(* IEC 61131-3 sources: CodesysTest/export/SX_1195.dev/Plc Logic/Application/PRJ Specific/Motion/Motors/Oriental AZD/AZD-KR2D/FB_OrientalAZMotorTriggerPositionTest.pou, 3 files *)

(* ---- FB_OrientalAZMotorTriggerPositionTest.pou.st ---- *)
(*#-#-#-#-#-#-#-#-#-#---Declaration---#-#-#-#-#-#-#-#-#-#-#-#-#*)

FUNCTION_BLOCK FB_OrientalAZMotorTriggerPositionTest EXTENDS Axis_REF
VAR_INPUT
	// Set this flag if this motor is actually a group
	isGroup : BOOL;
	// Steps per inch of motion
	stepsPerInchSP : DINT := 3999;
	// At factory "zero" there can be an offset
	zeroOffset : REAL;
	// Jog motor forward command
	jogForwardCMD : BOOL;
	// Jog motor reverse command
	jogReverseCMD : BOOL;
	// Factory "zero" positon preset command
	positionPresetRequest : BOOL;
	// Free up motor command
	freeMotorRequest : BOOL;
	// Ref to Master Motor if group
	groupMotor0 : REFERENCE TO FB_OrientalAZMotorTriggerPositionTest;
	// Ref to Slave Motor if group
	groupMotor1 : REFERENCE TO FB_OrientalAZMotorTriggerPositionTest;
END_VAR
VAR_OUTPUT
	// Hex alarm code reported from AZ Drive
	alarmCode : DWORD;
	// Trigger direct data write through modbus
	triggerDDWriteNow : BOOL;
	// Trigger Remote I/O data write through modbus
	triggerRIOWriteNow : BOOL;
END_VAR
VAR
	directDataOp : sctOrientalDirectData;
	distanceFromDrive : uModbusDWORD;
	alarmCodeFromDrive : uModbusDWORD;
	ready : BOOL;
	alarmActive : BOOL;
	moving : BOOL;
	inPosition : BOOL;
	atTorqueLimit : BOOL;
	atPosition : BOOL;
	homeSwitchTrigger : BOOL;
	homeNow : BOOL;
	P_Preset : BOOL;
	start : BOOL;
	zHome : BOOL;
	stop : BOOL;
	freeMotor : BOOL;
	reset : BOOL;
	EL_Preset : BOOL;
	jogReverse : BOOL;
	jogForward : BOOL;
	packedRIO : uModbusDWORD;
	packedRIOLast : DWORD;
	delayTimer : Standard.TON := (PT := T#50MS);
	zHomeDelay : Standard.TON := (PT := T#250MS);
	presetDelay : Standard.TON := (PT := T#200MS);
	modbusWriteResponse : ARRAY[0..20] OF WORD;
	readAfterDDWrite : FB_ONS;
	readAfterRIOWrite : FB_ONS;
	triggerPositonPreset : FB_ONS;
	haltONS : FB_ONS;
	alarmActiveONS : FB_ONS;
	freeMotorRequestONS : FB_ONS;
	triggerRIOWrite : BOOL;
	resetRIOWrite : Standard.TON := (PT := T#50MS);
	disable : BOOL;
	enumAlarmCode : eOrientalAZDriveFaults;
	state : eOrientalAZDriveStates;
	nextState : eOrientalAZDriveStates;
	commErrorONS : FB_ONS;
	commErrorFaultONS : FB_ONS;
	commErrorCount : DINT;
	commErrorFaultSetting : DINT := 3;
	positionPresetONS : FB_ONS;
END_VAR
VAR_IN_OUT
	MBChannel : IoDrvModbus.ModbusSlaveComPort;
	modbusDataFromDrive : ARRAY[0..39] OF WORD;
	modbusDirectDataToDrive : ARRAY[0..16] OF WORD;
	modbusRIODataToDrive : ARRAY[0..1] OF WORD;
END_VAR(*#-#-#-#-#-#-#-#-#-#---Implementation---#-#-#-#-#-#-#-#-#-#-#-#-#*)

//	Function Block: FB_OrientalAZMotor()
//	Description: A PLCOpen Motion compliant library for a Oriental AZ Series drive/motor
//
//	Created by: Ben Hess
//	Created Date: Tuesday, June 2nd 2020

// Outputs for Motion Lib
operational := PowerOn;
EnableState := DriveEnable;

// Exit if drive isn't enabled.
IF NOT DriveEnable THEN
	Error := FALSE;
	RETURN;
END_IF

// Get raw drive position and alarm code
IF isGroup THEN
	IF __ISVALIDREF(groupMotor0) THEN
		actPos := groupMotor0.ActualPosition;
		enumAlarmCode := groupMotor0.enumAlarmCode;
	END_IF
ELSE
	distanceFromDrive.wWord[0] := modbusDataFromDrive[3];
	distanceFromDrive.wWord[1] := modbusDataFromDrive[2];
	actPos := (TO_REAL(distanceFromDrive.diDint) / TO_REAL(stepsPerInchSP)) + zeroOffset;
	alarmCodeFromDrive.wWord[0] := modbusDataFromDrive[7];
	alarmCodeFromDrive.wWord[1] := modbusDataFromDrive[6];
	enumAlarmCode := TO_INT(alarmCodeFromDrive.diDint);
END_IF
alarmCode := TO_DWORD(enumAlarmCode);

// Pack RIO to write to drive
packedRIO.dDword.0 := homeSwitchTrigger;
packedRIO.dDword.1 := homeNow;
packedRIO.dDword.2 := P_Preset;
packedRIO.dDword.3 := start;
packedRIO.dDword.4 := zHome;
packedRIO.dDword.5 := stop;
packedRIO.dDword.6 := freeMotor;
packedRIO.dDword.7 := reset;
packedRIO.dDword.12 := EL_Preset;
packedRIO.dDword.13 := jogReverse;
packedRIO.dDword.14 := jogForward;
modbusRIODataToDrive[0] := packedRIO.wWord[1];
modbusRIODataToDrive[1] := packedRIO.wWord[0];

// Setup delay timers
delayTimer(IN := state = eOrientalAZDriveStates.DelayAfterWrite);
zHomeDelay(IN := state = eOrientalAZDriveStates.Homing);
presetDelay(IN := state = eOrientalAZDriveStates.SettingPreset);
// Trigger an RIO write whenever it changes
IF packedRIO.dDword <> packedRIOLast AND NOT triggerRIOWriteNow THEN
	packedRIOLast := packedRIO.dDword;
	triggerRIOWriteNow := TRUE;
END_IF
resetRIOWrite(IN := triggerRIOWriteNow);
IF resetRIOWrite.Q THEN
	triggerRIOWriteNow := FALSE;
END_IF
positionPresetONS(CLK := positionPresetRequest);

// Only set comm error status after x modbus errors
commErrorONS(CLK := MBChannel.xError);
IF commErrorONS.OSR THEN
	commErrorCount := commErrorCount + 1;
END_IF
commErrorFaultONS(CLK := commErrorCount = commErrorFaultSetting);
IF NOT isGroup THEN
	IF commErrorFaultONS.OSR THEN
		state := eOrientalAZDriveStates.Faulting;
		CommStatus := FALSE;
	END_IF
END_IF

// Get drive data directly from modbus or from master axis
IF isGroup THEN
	IF __ISVALIDREF(groupMotor0) AND __ISVALIDREF(groupMotor1) THEN
		ready := groupMotor0.ready AND groupMotor1.ready;
		alarmActive := groupMotor0.alarmActive OR groupMotor1.alarmActive;
		moving := groupMotor0.moving AND groupMotor1.moving;
		inPosition := groupMotor0.inPosition AND groupMotor1.inPosition;
		atTorqueLimit := groupMotor0.atTorqueLimit OR groupMotor1.atTorqueLimit;
	END_IF
ELSE
	Ready := modbusDataFromDrive[5].5;
	AlarmActive := modbusDataFromDrive[5].7;
	Moving := modbusDataFromDrive[5].13;
	InPosition := modbusDataFromDrive[5].14;
	AtTorqueLimit := modbusDataFromDrive[5].15;
END_IF

// Halt motor when Halt command seen
haltONS(CLK := Halt);
IF haltONS.OSR THEN
	state := eOrientalAZDriveStates.Halt;
END_IF

triggerPositonPreset(CLK := positionPresetRequest);
freeMotorRequestONS(CLK := freeMotorRequest);

// Reset motor when AckError command seen
IF AckError THEN
	state := eOrientalAZDriveStates.Resetting;
END_IF
alarmActiveONS(clk:= alarmActive);
IF alarmActiveONS.OSR THEN
	state := eOrientalAZDriveStates.Faulting;
END_IF

// Main motor state machine
CASE state OF
	eOrientalAZDriveStates.Idle:

				// 	Idle state, wait for command
				IF MoveAbs THEN
					freeMotor := FALSE;
					TargetReached := FALSE;
					AxisState := eAxisState.DiscreteMotion;
					state := eOrientalAZDriveStates.MoveABS;
				ELSIF MoveRel THEN
					freeMotor := FALSE;
					TargetReached := FALSE;
					AxisState := eAxisState.DiscreteMotion;
					state := eOrientalAZDriveStates.MoveInc;
				ELSIF MoveAbsTorque THEN
					freeMotor := FALSE;
					TargetReached := FALSE;
					AxisState := eAxisState.DiscreteMotion;
					state := eOrientalAZDriveStates.MovePush;
				ELSIF jogForwardCMD OR jogReverseCMD THEN
					state := eOrientalAZDriveStates.Jogging;
				ELSIF StartHoming THEN
					freeMotor := FALSE;
					isHomed := FALSE;
					//AxisState := AXIS_STATE.AS_Homing;
					state := eOrientalAZDriveStates.Home;
				ELSIF triggerPositonPreset.OSR THEN
					state := eOrientalAZDriveStates.SetPreset;
				END_IF
				IF MBChannel.xDone OR isGroup THEN
					CommStatus := TRUE;
					commErrorCount := 0;
				END_IF

	eOrientalAZDriveStates.MoveABS:
				// Move to absolute position
				directDataOp.OperationType.diDint := eOrientalOperationType.Absolute_Positioning;
				directDataOp.Position.diDint := mDistanceCalc(targetPosDist);
				directDataOp.Speed.diDint := mVeloAccDecCalc(ProfileVelocity);
				directDataOp.RateOfChange.diDint := mVeloAccDecCalc(ProfileAcceleration);
				directDataOp.StoppingDecel.diDint := mVeloAccDecCalc(ProfileDeceleration);
				directDataOp.Current.diDint := mCurrentCalc(DefaultCurrent);
				directDataOp.Trigger.diDint := 1;
				mPackDDOp();
				triggerDDWriteNow := TRUE;
				state := eOrientalAZDriveStates.DelayAfterWrite;
				nextState := eOrientalAZDriveStates.Moving;

	eOrientalAZDriveStates.MovePush:
				// Move to absolute position "push" (at a limited current)
				directDataOp.OperationType.diDint := eOrientalOperationType.Absolute_Push;
				directDataOp.Position.diDint := mDistanceCalc(targetPosDist);
				directDataOp.Speed.diDint := mVeloAccDecCalc(ProfileVelocity);
				directDataOp.RateOfChange.diDint := mVeloAccDecCalc(ProfileAcceleration);
				directDataOp.StoppingDecel.diDint := mVeloAccDecCalc(ProfileDeceleration);
				directDataOp.Current.diDint := mCurrentCalc(ProfileCurrentLimit);
				directDataOp.Trigger.diDint := 1;
				mPackDDOp();
				triggerDDWriteNow := TRUE;

				state := eOrientalAZDriveStates.DelayAfterWrite;
				nextState := eOrientalAZDriveStates.Moving;

		eOrientalAZDriveStates.MoveInc:

				// Move to incremental position
				directDataOp.OperationType.diDint := eOrientalOperationType.Incremental_Positioning;
				directDataOp.Position.diDint := mDistanceCalc(targetPosDist);
				directDataOp.Speed.diDint := mVeloAccDecCalc(ProfileVelocity);
				directDataOp.RateOfChange.diDint := mVeloAccDecCalc(ProfileAcceleration);
				directDataOp.StoppingDecel.diDint := mVeloAccDecCalc(ProfileDeceleration);
				directDataOp.Current.diDint := mCurrentCalc(DefaultCurrent);
				directDataOp.Trigger.diDint := 1;
				mPackDDOp();
				triggerDDWriteNow := TRUE;

				state := eOrientalAZDriveStates.DelayAfterWrite;
				nextState := eOrientalAZDriveStates.Moving;

		eOrientalAZDriveStates.Home:
				// Home motor
				zHome := TRUE;
				state := eOrientalAZDriveStates.DelayAfterWrite;
				nextState := eOrientalAZDriveStates.Homing;

		eOrientalAZDriveStates.Homing:
				// Wait until ZHome is done
				IF zHomeDelay.Q AND TO_DINT(actPos * 1000) >= (TO_DINT(zeroOffset * 1000) - 10) AND TO_DINT(actPos * 1000) <= (TO_DINT(zeroOffset * 1000) + 10) THEN
					zHome := FALSE;
					isHomed := TRUE;
					state := eOrientalAZDriveStates.DoneMoving;
				END_IF

		eOrientalAZDriveStates.Jogging:
				// Jog forward/reverse
				jogForward := jogForwardCMD;
				jogReverse := jogReverseCMD;

				IF NOT jogForward AND NOT jogReverse THEN
					state := eOrientalAZDriveStates.Idle;
				END_IF

		eOrientalAZDriveStates.SetPreset:
				// Set factory ZERO preset
				freeMotor := TRUE;
				//P_Preset := TRUE;
				IF triggerPositonPreset.OSF THEN
					state := eOrientalAZDriveStates.SettingPreset;
				END_IF

		eOrientalAZDriveStates.SettingPreset:
				// Set factory zero preset on AZ Motor
				P_Preset := TRUE;
				IF distanceFromDrive.dDword = 0 OR presetDelay.Q THEN
					freeMotor := FALSE;
					P_Preset := FALSE;
					state := eOrientalAZDriveStates.Idle;
				END_IF

		eOrientalAZDriveStates.SetPresetDone:
				//
		eOrientalAZDriveStates.DelayAfterWrite:
				// A small delay before moving on to next state
				IF delayTimer.Q THEN
					triggerDDWriteNow := FALSE;
					state := nextState;
				END_IF

		eOrientalAZDriveStates.Moving:
				// After sending data, we are moving
				IF (mInPosition() AND (MoveAbs OR MoveAbsTorque)) OR (atTorqueLimit AND MoveAbsTorque) OR (inPosition AND MoveRel) THEN
					TargetReached := TRUE;
					state := eOrientalAZDriveStates.DoneMoving;
				END_IF

		eOrientalAZDriveStates.DoneMoving:
				// Wait for status to clear
				IF NOT MoveAbs AND NOT MoveAbsTorque AND NOT MoveRel AND NOT StartHoming THEN
					AxisState := eAxisState.Standstill;
					state := eOrientalAZDriveStates.Idle;
				END_IF

		eOrientalAZDriveStates.Halt:
				//
				freeMotor := TRUE;
				AxisState := eAxisState.ErrorStop;
				state := eOrientalAZDriveStates.Halted;

		eOrientalAZDriveStates.Halted:
				//
				IF AckError THEN
					state := eOrientalAZDriveStates.Resetting;
					freeMotor := FALSE;
				END_IF

		eOrientalAZDriveStates.Faulting:
				// Faulting - stop drive
				mClearStatus();
				AxisState := eAxisState.ErrorStop;
				Error := TRUE;
				freeMotor := TRUE;
				zHome := FALSE;
				//triggerRIOWriteNow := TRUE;
				state := eOrientalAZDriveStates.Faulted;

		eOrientalAZDriveStates.Faulted:
				// Faulted - wait for clear
				IF AckError THEN
					state := eOrientalAZDriveStates.Resetting;
				END_IF

		eOrientalAZDriveStates.Resetting:
				//
					CommStatus := TRUE;
					commErrorCount := 0;
					IF alarmActive THEN
						reset := TRUE;
					END_IF
					IF NOT alarmActive THEN
						triggerDDWriteNow := FALSE;
						triggerRIOWriteNow := FALSE;
						AckError := FALSE;
						Error := FALSE;
						freeMotor := FALSE;
						reset := FALSE;
						zHome := FALSE;
						MoveAbs := FALSE;
						MoveRel := FALSE;
						MoveAbsTorque := FALSE;
						StartHoming := FALSE;
						state := eOrientalAZDriveStates.Idle;
						nextState := eOrientalAZDriveStates.Idle;
					END_IF
END_CASE

(* ---- mDistanceCalc.m.st ---- *)
(*#-#-#-#-#-#-#-#-#-#---Declaration---#-#-#-#-#-#-#-#-#-#-#-#-#*)

METHOD PRIVATE mDistanceCalc : DINT
VAR_INPUT
	distanceSP : REAL;
END_VAR
(*#-#-#-#-#-#-#-#-#-#---Implementation---#-#-#-#-#-#-#-#-#-#-#-#-#*)

IF directDataOp.OperationType.diDint = eOrientalOperationType.Absolute_Positioning OR directDataOp.OperationType.diDint = eOrientalOperationType.Absolute_Push THEN
	mDistanceCalc := TO_DINT((distanceSP - zeroOffset) * TO_REAL(stepsPerInchSP));
ELSE
	mDistanceCalc := TO_DINT((distanceSP) * TO_REAL(stepsPerInchSP));
END_IF

(* ---- mInPosition.m.st ---- *)
(*#-#-#-#-#-#-#-#-#-#---Declaration---#-#-#-#-#-#-#-#-#-#-#-#-#*)

METHOD PRIVATE mInPosition : BOOL
VAR_INPUT
END_VAR
(*#-#-#-#-#-#-#-#-#-#---Implementation---#-#-#-#-#-#-#-#-#-#-#-#-#*)

// Set in position status if we're float =
mInPosition := TO_DINT(actPos * 1000) >= (TO_DINT(targetPosDist * 1000) - 10) AND TO_DINT(actPos * 1000) <= (TO_DINT(targetPosDist * 1000) + 10);
